(****************************************************************
NAME:			FB_Move
DATA:			2017.2.17
VERSION:		1.0.0
DESCRIPTION:	FB_Move
HISTORY:
				2017.2.17		NEW
				2018.1.9		ÐÂÔöBCGapMode
***************************************************************)
FUNCTION_BLOCK FB_Move
VAR_INPUT
	(*È«¾Ö*)
	Mode:DINT;
	PowerState:BOOL;
	(*BCGapMode*)
	TargetGapPosition:LREAL;
	TargetGapVelocity:LREAL;
	BCGapMove:BOOL;
	BCGapReset:BOOL;
END_VAR
VAR_OUTPUT
	FbID:DINT:=1001;

	BCGapState:DINT;
	BCGapBusy:BOOL;
	BCGapDone:BOOL;
	GapMoving:BOOL;
	Error:BOOL;
	ErrorID:DINT;
END_VAR
VAR
	PhaseShifterLin_MC_MoveAbsolute: MC_MoveAbsolute;
	fb_ton: TON;
	fb_ton1: TON;
	fb_ton2: TON;
	fb_ton_debug_1:TON;
	fb_ton_debug_2:TON;
	fb_ton_debug_3:TON;
	fb_ton_debug_4:TON;
	fb_ton_BC:TON;
	fb_ton_BC_2:TON;
	
END_VAR

IF PowerState=1 THEN
	IF Mode=1 AND BCGapMove THEN
		A_BCGapMove();
	END_IF
END_IF

ACTION A_BCGapMove:
IF BCGapMove THEN
	BCGapBusy:=TRUE;
	BCGapDone:=FALSE;
	fb_ton_BC(PT:=t#80s);(*2mm/s max spees,120mmÐÐ³Ì£¬60sÄÚ×ßÍê*)
	A_MoveMC();
	IF  PhaseShifterLin.Status.Moving  THEN
		GapMoving:=TRUE;
	ELSE
		GapMoving:=FALSE;
	END_IF
	CASE BCGapState OF
		0:
			IF PhaseShifterLin.Status.Moving THEN	(*ÖáÕýÔÚÔËÐÐ£¬Ñ­»·¸Ã²½µÈ´ý*)
				BCGapState:=88;
			ELSIF PhaseShifterLin.Status.NotMoving THEN	(*Öá¶¼´¦ÓÚÍ£Ö¹×´Ì¬Ê±£¬×ªÏÂÒ»²½*)
				BCGapState:=1;
			END_IF
		1:
			PhaseShifterLin_MC_MoveAbsolute.Position:=TargetGapPosition;
			PhaseShifterLin_MC_MoveAbsolute.Velocity:=TargetGapVelocity;
			PhaseShifterLin_MC_MoveAbsolute.Execute:=TRUE;
			fb_ton_BC.IN:=TRUE;
			BCGapState:=2;
		2:
			IF NOT PhaseShifterLin_MC_MoveAbsolute.Done THEN		(*ÔË¶¯ÖÐ£¬¼ì²éDoneÐÅºÅ£¬Ã»ÓÐÔòÑ­»·*)
				BCGapState:=2;
			ELSIF PhaseShifterLin_MC_MoveAbsolute.Done THEN		(*ÔË¶¯Íê³É£¬×ªÏÂÒ»²½*)
				BCGapState:=88;
			END_IF
	
		88:
			BCGapMove:=FALSE;
			BCGapState:=0;
			BCGapBusy:=FALSE;
			BCGapDone:=TRUE;
			Error:=FALSE;
			ErrorID:=0;
			PhaseShifterLin_MC_MoveAbsolute.Execute:=FALSE;
			fb_ton_BC.IN:=FALSE;
		89:
			BCGapMove:=FALSE;
			BCGapState:=0;
			BCGapBusy:=FALSE;
			BCGapDone:=FALSE;
			Error:=FALSE;
			ErrorID:=0;
			PhaseShifterLin_MC_MoveAbsolute.Execute:=FALSE;
			fb_ton_BC.IN:=FALSE;
		99:
			BCGapMove:=FALSE;
			BCGapState:=99;
			BCGapBusy:=FALSE;
			BCGapDone:=FALSE;
			Error:=TRUE;
			PhaseShifterLin_MC_MoveAbsolute.Execute:=FALSE;
			fb_ton_BC.IN:=FALSE;
		-100:
			FB_PlcEmergencyStop();
			BCGapMove:=FALSE;
			BCGapState:=-100;
			BCGapBusy:=FALSE;
			BCGapDone:=FALSE;
			Error:=TRUE;
			PhaseShifterLin_MC_MoveAbsolute.Execute:=FALSE;
			fb_ton_BC.IN:=FALSE;
	END_CASE
	IF BCGapReset THEN
		BCGapReset:=FALSE;
		BCGapMove:=FALSE;
		BCGapState:=0;
		BCGapBusy:=FALSE;
		BCGapDone:=FALSE;
		Error:=FALSE;
		ErrorID:=0;
		PhaseShifterLin_MC_MoveAbsolute.Execute:=FALSE;
		fb_ton_BC.IN:=FALSE;
	END_IF
END_IF
END_ACTION

ACTION A_MoveMC:
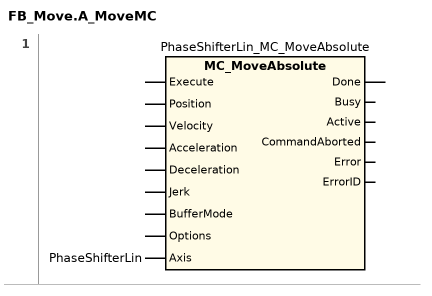
// NETWORK 1
PhaseShifterLin_MC_MoveAbsolute(Axis := PhaseShifterLin); // MC_MoveAbsolute
END_ACTION

END_FUNCTION_BLOCK

(* stored: Version 1.1.0.1, ProductVersion 3.1.4024.6
   POU FB_Move: Id {f9a99ade-b4af-4565-bffe-bba1640e411e}, SpecialFunc None
   Action A_BCGapMove: Id {14a23b8d-1d11-4027-a881-ef621e956d3f}
   Action A_MoveMC: Id {f577884c-c19e-4448-8f5c-62de64b66e2f} *)
